# EPICS substitutions: tgpApp/Db/TPG366.substitutions
# Mandatory macros:
# CONTROLLER  Name of the MaxiGauge (PV prefix)
# PORT        Asyn port of the MaxiGauge

# In the following macro names x stands for 1...6 (per channel) or _ (all channels)
# Optional macros:
# ADDR        address 1-9 (default: 1, ignored when connected to TCP network)
# SENSORx     Names of the vacuum sensors, default to $(CONTROLLER)-SENSORx
# P,Sx        Shortcuts for SENSORx: $(SENSORx)=$(P)$(Sx)
# WARNx       MINOR alarm level, defaults Inf (no warning)
# ALARMx      MAJOR alarm level, defaults Inf (no alarm)
# MINx        Minimal range exponent, defaults to -11
# MAXx        Maximal range exponent, defaults to 3
# PRECx       Precision, defaults to -4 (4 digit exponential)
# ASG         Access Security Group, defaults to ""
# FASTSCAN    Scanrate for pressure etc, defaults to "1 second"
# SLOWSCAN    Scanrate for sensor names etc, defaults to "10 second"

file TPG366-Sensor.template
{ pattern
  {CH    SENSOR                                        PREC                   MIN                  MAX                   WARN                    ALARM                   }
  { 1 "$(SENSOR1=$(P=$(CONTROLLER)-)$(S1=SENSOR1))" "$(PREC1=$(PREC_=-4))" "$(MIN1=$(MIN_=-11))" "$(MAX1=$(MAX_=3))" "$(WARN1=$(WARN_=Inf))" "$(ALARM1=$(ALARM_=Inf))" }
  { 2 "$(SENSOR2=$(P=$(CONTROLLER)-)$(S2=SENSOR2))" "$(PREC2=$(PREC_=-4))" "$(MIN2=$(MIN_=-11))" "$(MAX2=$(MAX_=3))" "$(WARN2=$(WARN_=Inf))" "$(ALARM2=$(ALARM_=Inf))" }
  { 3 "$(SENSOR3=$(P=$(CONTROLLER)-)$(S3=SENSOR3))" "$(PREC3=$(PREC_=-4))" "$(MIN3=$(MIN_=-11))" "$(MAX3=$(MAX_=3))" "$(WARN3=$(WARN_=Inf))" "$(ALARM3=$(ALARM_=Inf))" }
  { 4 "$(SENSOR4=$(P=$(CONTROLLER)-)$(S4=SENSOR4))" "$(PREC4=$(PREC_=-4))" "$(MIN4=$(MIN_=-11))" "$(MAX4=$(MAX_=3))" "$(WARN4=$(WARN_=Inf))" "$(ALARM4=$(ALARM_=Inf))" }
  { 5 "$(SENSOR5=$(P=$(CONTROLLER)-)$(S5=SENSOR5))" "$(PREC5=$(PREC_=-4))" "$(MIN5=$(MIN_=-11))" "$(MAX5=$(MAX_=3))" "$(WARN5=$(WARN_=Inf))" "$(ALARM5=$(ALARM_=Inf))" }
  { 6 "$(SENSOR6=$(P=$(CONTROLLER)-)$(S6=SENSOR6))" "$(PREC6=$(PREC_=-4))" "$(MIN6=$(MIN_=-11))" "$(MAX6=$(MAX_=3))" "$(WARN6=$(WARN_=Inf))" "$(ALARM6=$(ALARM_=Inf))" }
}

file TPG366-Setpoint.template
{ pattern
  {NR NRC    PREC}
  {1   A  "$(PRECA=$(PRECSP=$(PREC_=-4)))" }
  {2   B  "$(PRECB=$(PRECSP=$(PREC_=-4)))" }
  {3   C  "$(PRECC=$(PRECSP=$(PREC_=-4)))" }
  {4   D  "$(PRECD=$(PRECSP=$(PREC_=-4)))" }
  {5   E  "$(PRECE=$(PRECSP=$(PREC_=-4)))" }
  {6   F  "$(PRECF=$(PRECSP=$(PREC_=-4)))" }
}
